ABB RAPID module: Module1.mod

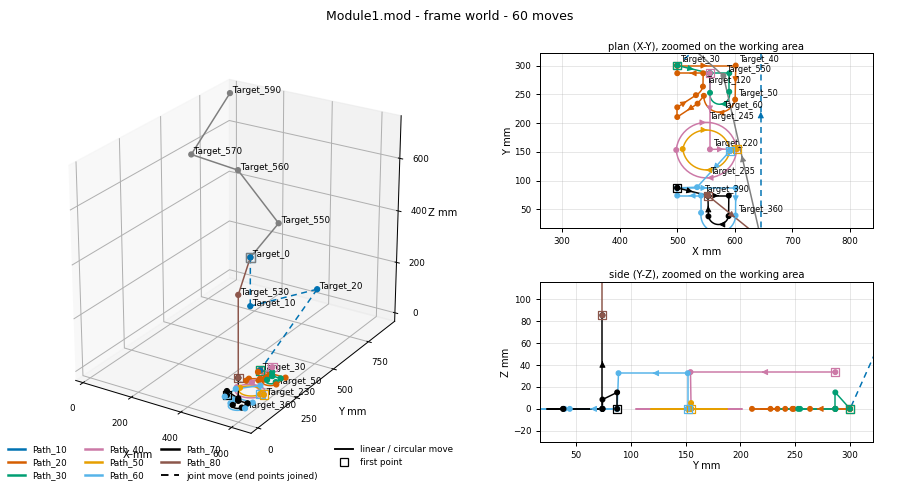
[picture p0: tool path of Module1.mod in frame world, 60 of 60 moves have a stored position in this frame; points joined in program order, loops and branches not executed]
MODULE Module1
    CONST robtarget Target_0:=[[145.114046101,-300,573.947441117],[0.5,0,0.866025404,0],[0,0,0,0],[9E+09,9E+09,9E+09,9E+09,9E+09,9E+09]];
    CONST robtarget Target_10:=[[145.11412777,-300,402.018378698],[0.500000003,0,0.866025402,0],[0,0,0,0],[9E+09,9E+09,9E+09,9E+09,9E+09,9E+09]];
    CONST robtarget Target_20:=[[145.114134181,130.918790149,291.07357],[0.500000009,0.000000018,0.866025398,-0.00000003],[0,-1,1,0],[9E+09,9E+09,9E+09,9E+09,9E+09,9E+09]];
    CONST robtarget Target_30:=[[0,0,0],[0,1,0,0],[0,0,-2,0],[9E+09,9E+09,9E+09,9E+09,9E+09,9E+09]];
    CONST robtarget Target_40:=[[101.558,0,0],[0,1,0,0],[0,0,-2,0],[9E+09,9E+09,9E+09,9E+09,9E+09,9E+09]];
    CONST robtarget Target_50:=[[100.559,-59.146,0],[0,1,0,0],[0,0,-2,0],[9E+09,9E+09,9E+09,9E+09,9E+09,9E+09]];
    CONST robtarget Target_60:=[[73.842,-81.151,0],[0,1,0,0],[0,0,-2,0],[9E+09,9E+09,9E+09,9E+09,9E+09,9E+09]];
    CONST robtarget Target_70:=[[46.206,-52.556,0],[0,1,0,0],[0,0,-2,0],[9E+09,9E+09,9E+09,9E+09,9E+09,9E+09]];
    CONST robtarget Target_80:=[[35.263,-66.215,0],[0,1,0,0],[0,0,-2,0],[9E+09,9E+09,9E+09,9E+09,9E+09,9E+09]];
    CONST robtarget Target_90:=[[-0.001,-89.458,0],[0,1,0,0],[0,0,-2,0],[9E+09,9E+09,9E+09,9E+09,9E+09,9E+09]];
    CONST robtarget Target_100:=[[-0.001,-72.564,0],[0,1,0,0],[0,0,-2,0],[9E+09,9E+09,9E+09,9E+09,9E+09,9E+09]];
    CONST robtarget Target_110:=[[32.467,-51.478,0],[0,1,0,0],[0,0,-2,0],[9E+09,9E+09,9E+09,9E+09,9E+09,9E+09]];
    CONST robtarget Target_115:=[[41.413,-43.371,0],[0,1,0,0],[0,0,-2,0],[9E+09,9E+09,9E+09,9E+09,9E+09,9E+09]];
    CONST robtarget Target_120:=[[44.608,-36.502,0],[0,1,0,0],[0,0,-2,0],[9E+09,9E+09,9E+09,9E+09,9E+09,9E+09]];
    CONST robtarget Target_130:=[[45.087,-13.418,0],[0,1,0,0],[0,0,-2,0],[9E+09,9E+09,9E+09,9E+09,9E+09,9E+09]];
    CONST robtarget Target_140:=[[-0.001,-13.418,0],[0,1,0,0],[0,0,-2,0],[9E+09,9E+09,9E+09,9E+09,9E+09,9E+09]];
    CONST robtarget Target_145:=[[0,0,0],[0,1,0,0],[0,0,-2,0],[9E+09,9E+09,9E+09,9E+09,9E+09,9E+09]];
    CONST robtarget Target_150_IntermedioR:=[[56.636379342,-13.418007291,15.010665058],[-0.000000015,1,0.000000042,0.000000001],[0,0,-2,0],[9E+09,9E+09,9E+09,9E+09,9E+09,9E+09]];
    CONST robtarget Target_150_ZFinal:=[[56.749,-13.418,0],[0,1,0,0],[0,0,-2,0],[9E+09,9E+09,9E+09,9E+09,9E+09,9E+09]];
    CONST robtarget Target_160:=[[90.336,-13.418,0],[0,1,0,0],[0,0,-2,0],[9E+09,9E+09,9E+09,9E+09,9E+09,9E+09]];
    CONST robtarget Target_170:=[[90.336,-45.567,0],[0,1,0,0],[0,0,-2,0],[9E+09,9E+09,9E+09,9E+09,9E+09,9E+09]];
    CONST robtarget Target_180:=[[73.842,-67.293,0],[0,1,0,0],[0,0,-2,0],[9E+09,9E+09,9E+09,9E+09,9E+09,9E+09]];
    CONST robtarget Target_190:=[[56.909,-47.325,0],[0,1,0,0],[0,0,-2,0],[9E+09,9E+09,9E+09,9E+09,9E+09,9E+09]];
    CONST robtarget Target_200:=[[56.749,-13.418,0],[0,1,0,0],[0,0,-2,0],[9E+09,9E+09,9E+09,9E+09,9E+09,9E+09]];
    CONST robtarget Target_210:=[[56.748968334,-13.418012212,33.529365391],[-0.000000004,1,-0.000000052,-0.000000031],[0,0,-2,0],[9E+09,9E+09,9E+09,9E+09,9E+09,9E+09]];
    CONST robtarget Target_220:=[[56.748986906,-145.605410925,33.52934752],[0,1,-0.000000083,-0.000000019],[0,0,-2,0],[9E+09,9E+09,9E+09,9E+09,9E+09,9E+09]];
    CONST robtarget Target_230:=[[103.355,-145.049,0],[0,1,0,0],[0,0,-2,0],[9E+09,9E+09,9E+09,9E+09,9E+09,9E+09]];
    CONST robtarget Target_235:=[[52.116,-195.19,0],[0,1,0,0],[0,0,-2,0],[9E+09,9E+09,9E+09,9E+09,9E+09,9E+09]];
    CONST robtarget Target_240:=[[-1.758,-146.687,0],[0,1,0,0],[0,0,-2,0],[9E+09,9E+09,9E+09,9E+09,9E+09,9E+09]];
    CONST robtarget Target_245:=[[50.261,-98.729,0],[0,1,0,0],[0,0,-2,0],[9E+09,9E+09,9E+09,9E+09,9E+09,9E+09]];
    CONST robtarget Target_250:=[[103.355,-145.049,0],[0,1,0,0],[0,0,-2,0],[9E+09,9E+09,9E+09,9E+09,9E+09,9E+09]];
    CONST robtarget Target_260:=[[97.170116811,-145.0489929,5.322039607],[0.000000004,1,0.000000037,0.000000006],[0,-1,-2,0],[9E+09,9E+09,9E+09,9E+09,9E+09,9E+09]];
    CONST robtarget Target_270:=[[91.773,-147.965,0],[0,1,0,0],[0,0,-2,0],[9E+09,9E+09,9E+09,9E+09,9E+09,9E+09]];
    CONST robtarget Target_280:=[[48.761,-181.312,0],[0,1,0,0],[0,0,-2,0],[9E+09,9E+09,9E+09,9E+09,9E+09,9E+09]];
    CONST robtarget Target_290:=[[9.487,-145.045,0],[0,1,0,0],[0,0,-2,0],[9E+09,9E+09,9E+09,9E+09,9E+09,9E+09]];
    CONST robtarget Target_300:=[[50.519,-112.002,0],[0,1,0,0],[0,0,-2,0],[9E+09,9E+09,9E+09,9E+09,9E+09,9E+09]];
    CONST robtarget Target_310:=[[91.935,-148.087,0],[0,1,0,0],[0,0,-2,0],[9E+09,9E+09,9E+09,9E+09,9E+09,9E+09]];
    CONST robtarget Target_320:=[[91.93496497,-148.087005279,32.547397703],[0.000000003,1,0.000000045,-0.000000008],[0,-1,-2,0],[9E+09,9E+09,9E+09,9E+09,9E+09,9E+09]];
    CONST robtarget Target_330:=[[34.441170169,-211.299624395,32.547366159],[-0.000000002,1,0.000000004,-0.000000023],[0,0,-2,0],[9E+09,9E+09,9E+09,9E+09,9E+09,9E+09]];
    CONST robtarget Target_340:=[[-0.001,-212.542,0],[0,1,0,0],[0,0,-2,0],[9E+09,9E+09,9E+09,9E+09,9E+09,9E+09]];
    CONST robtarget Target_350:=[[101.558,-212.542,0],[0,1,0,0],[0,0,-2,0],[9E+09,9E+09,9E+09,9E+09,9E+09,9E+09]];
    CONST robtarget Target_360:=[[101.278,-260.506,0],[0,1,0,0],[0,0,-2,0],[9E+09,9E+09,9E+09,9E+09,9E+09,9E+09]];
    CONST robtarget Target_370:=[[72.204,-290.019,0],[0,1,0,0],[0,0,-2,0],[9E+09,9E+09,9E+09,9E+09,9E+09,9E+09]];
    CONST robtarget Target_380:=[[41.373,-255.754,0],[0,1,0,0],[0,0,-2,0],[9E+09,9E+09,9E+09,9E+09,9E+09,9E+09]];
    CONST robtarget Target_390:=[[41.293,-225.961,0],[0,1,0,0],[0,0,-2,0],[9E+09,9E+09,9E+09,9E+09,9E+09,9E+09]];
    CONST robtarget Target_400:=[[-0.001,-225.961,0],[0,1,0,0],[0,0,-2,0],[9E+09,9E+09,9E+09,9E+09,9E+09,9E+09]];
    CONST robtarget Target_410:=[[-0.001,-212.542,0],[0,1,0,0],[0,0,-2,0],[9E+09,9E+09,9E+09,9E+09,9E+09,9E+09]];
    CONST robtarget Target_420:=[[-0.00102366,-212.542012413,15.028104182],[-0.000000001,1,-0.000000059,-0.000000007],[0,0,-2,0],[9E+09,9E+09,9E+09,9E+09,9E+09,9E+09]];
    CONST robtarget Target_430:=[[53.40676855,-225.942037535,8.490466142],[-0.000000001,1,-0.000000385,-0.000000007],[0,0,-2,0],[9E+09,9E+09,9E+09,9E+09,9E+09,9E+09]];
    CONST robtarget Target_440:=[[53.274,-225.961,0],[0,1,0,0],[0,0,-2,0],[9E+09,9E+09,9E+09,9E+09,9E+09,9E+09]];
    CONST robtarget Target_450:=[[89.577,-225.961,0],[0,1,0,0],[0,0,-2,0],[9E+09,9E+09,9E+09,9E+09,9E+09,9E+09]];
    CONST robtarget Target_460:=[[89.177,-261.505,0],[0,1,0,0],[0,0,-2,0],[9E+09,9E+09,9E+09,9E+09,9E+09,9E+09]];
    CONST robtarget Target_470:=[[71.765,-276.161,0],[0,1,0,0],[0,0,-2,0],[9E+09,9E+09,9E+09,9E+09,9E+09,9E+09]];
    CONST robtarget Target_480:=[[54.153,-261.984,0],[0,1,0,0],[0,0,-2,0],[9E+09,9E+09,9E+09,9E+09,9E+09,9E+09]];
    CONST robtarget Target_490:=[[53.274,-225.961,0],[0,1,0,0],[0,0,-2,0],[9E+09,9E+09,9E+09,9E+09,9E+09,9E+09]];
    CONST robtarget Target_500:=[[53.273969687,-225.961003513,85.391501657],[-0.000000001,1,0.000000011,-0.000000007],[0,0,-2,0],[9E+09,9E+09,9E+09,9E+09,9E+09,9E+09]];
    CONST robtarget Target_530:=[[53.273975183,-225.961003543,389.504685045],[0.000000001,1,0.000000014,-0.000000011],[0,0,-2,0],[9E+09,9E+09,9E+09,9E+09,9E+09,9E+09]];
    CONST robtarget Target_540:=[[145.114046101,-300,573.947441117],[0.5,0,0.866025404,0],[0,0,0,0],[9E+09,9E+09,9E+09,9E+09,9E+09,9E+09]];
    CONST robtarget Target_550:=[[80.158887002,-17.886905109,573.947441117],[0.487251492,-0.194314053,0.84394434,0.112187271],[0,0,0,0],[9E+09,9E+09,9E+09,9E+09,9E+09,9E+09]];
    CONST robtarget Target_560:=[[-281.152242484,306.8589552,573.947441117],[0.409151388,-0.497780499,0.708670992,0.287393705],[0,-1,-1,0],[9E+09,9E+09,9E+09,9E+09,9E+09,9E+09]];
    CONST robtarget Target_570:=[[-500.572509967,345.113792062,573.947441117],[0.353396474,-0.612644102,0.612100649,0.353710237],[1,-1,0,0],[9E+09,9E+09,9E+09,9E+09,9E+09,9E+09]];
    CONST robtarget Target_590:=[[-500.801741318,603.468233425,725.305628398],[0.499667188,-0.50033274,0.499889039,0.500110787],[1,-1,0,0],[9E+09,9E+09,9E+09,9E+09,9E+09,9E+09]];
    PROC Path_10()
        MoveJ Target_0,v1000,z10,ChuislitoToolTCP\WObj:=TablaPlana;
        MoveJ Target_10,v1000,z10,ChuislitoToolTCP\WObj:=TablaPlana;
        MoveJ Target_20,v1000,z10,ChuislitoToolTCP\WObj:=TablaPlana;
        MoveJ Target_30,v1000,z10,ChuislitoToolTCP\WObj:=TablaPlana;
    ENDPROC
    PROC Path_20()
        MoveL Target_30,v100,z5,ChuislitoToolTCP\WObj:=TablaPlana;
        MoveL Target_40,v100,z5,ChuislitoToolTCP\WObj:=TablaPlana;
        MoveL Target_50,v100,z5,ChuislitoToolTCP\WObj:=TablaPlana;
        MoveC Target_60,Target_70,v100,z5,ChuislitoToolTCP\WObj:=TablaPlana;
        MoveL Target_80,v100,z5,ChuislitoToolTCP\WObj:=TablaPlana;
        MoveL Target_90,v100,z5,ChuislitoToolTCP\WObj:=TablaPlana;
        MoveL Target_100,v100,z5,ChuislitoToolTCP\WObj:=TablaPlana;
        MoveL Target_110,v100,z5,ChuislitoToolTCP\WObj:=TablaPlana;
        MoveC Target_115,Target_120,v100,z5,ChuislitoToolTCP\WObj:=TablaPlana;
        MoveL Target_130,v100,z5,ChuislitoToolTCP\WObj:=TablaPlana;
        MoveL Target_140,v100,z5,ChuislitoToolTCP\WObj:=TablaPlana;
        MoveL Target_145,v100,z5,ChuislitoToolTCP\WObj:=TablaPlana;
    ENDPROC
    PROC Path_30()
        MoveL Target_145,v100,z5,ChuislitoToolTCP\WObj:=TablaPlana;
        MoveL Target_150_IntermedioR,v100,z5,ChuislitoToolTCP\WObj:=TablaPlana;
        MoveL Target_150_ZFinal,v100,z5,ChuislitoToolTCP\WObj:=TablaPlana;
        MoveL Target_160,v100,z5,ChuislitoToolTCP\WObj:=TablaPlana;
        MoveL Target_170,v100,z5,ChuislitoToolTCP\WObj:=TablaPlana;
        MoveC Target_180,Target_190,v100,z5,ChuislitoToolTCP\WObj:=TablaPlana;
        MoveL Target_200,v100,z5,ChuislitoToolTCP\WObj:=TablaPlana;
    ENDPROC
    PROC Path_40()
        MoveL Target_210,v100,z5,ChuislitoToolTCP\WObj:=TablaPlana;
        MoveL Target_220,v100,z5,ChuislitoToolTCP\WObj:=TablaPlana;
        MoveL Target_230,v100,z5,ChuislitoToolTCP\WObj:=TablaPlana;
        MoveC Target_235,Target_240,v100,z5,ChuislitoToolTCP\WObj:=TablaPlana;
        MoveC Target_245,Target_250,v100,z5,ChuislitoToolTCP\WObj:=TablaPlana;
    ENDPROC
    PROC Path_50()
        MoveL Target_250,v100,z5,ChuislitoToolTCP\WObj:=TablaPlana;
        MoveL Target_260,v100,z5,ChuislitoToolTCP\WObj:=TablaPlana;
        MoveL Target_270,v100,z5,ChuislitoToolTCP\WObj:=TablaPlana;
        MoveC Target_280,Target_290,v100,z5,ChuislitoToolTCP\WObj:=TablaPlana;
        MoveC Target_300,Target_310,v100,z5,ChuislitoToolTCP\WObj:=TablaPlana;
    ENDPROC
    PROC Path_60()
        MoveL Target_310,v100,z5,ChuislitoToolTCP\WObj:=TablaPlana;
        MoveL Target_320,v100,z5,ChuislitoToolTCP\WObj:=TablaPlana;
        MoveL Target_330,v100,z5,ChuislitoToolTCP\WObj:=TablaPlana;
        MoveL Target_340,v100,z5,ChuislitoToolTCP\WObj:=TablaPlana;
        MoveL Target_350,v100,z5,ChuislitoToolTCP\WObj:=TablaPlana;
        MoveL Target_360,v100,z5,ChuislitoToolTCP\WObj:=TablaPlana;
        MoveC Target_370,Target_380,v100,z5,ChuislitoToolTCP\WObj:=TablaPlana;
        MoveL Target_390,v100,z5,ChuislitoToolTCP\WObj:=TablaPlana;
        MoveL Target_400,v100,z5,ChuislitoToolTCP\WObj:=TablaPlana;
        MoveL Target_410,v100,z5,ChuislitoToolTCP\WObj:=TablaPlana;
    ENDPROC
    PROC Path_70()
        MoveL Target_410,v100,z5,ChuislitoToolTCP\WObj:=TablaPlana;
        MoveL Target_420,v100,z5,ChuislitoToolTCP\WObj:=TablaPlana;
        MoveL Target_430,v100,z5,ChuislitoToolTCP\WObj:=TablaPlana;
        MoveL Target_440,v100,z5,ChuislitoToolTCP\WObj:=TablaPlana;
        MoveL Target_450,v100,z5,ChuislitoToolTCP\WObj:=TablaPlana;
        MoveL Target_460,v100,z5,ChuislitoToolTCP\WObj:=TablaPlana;
        MoveC Target_470,Target_480,v100,z5,ChuislitoToolTCP\WObj:=TablaPlana;
        MoveL Target_490,v100,z5,ChuislitoToolTCP\WObj:=TablaPlana;
        MoveL Target_500,v100,z5,ChuislitoToolTCP\WObj:=TablaPlana;
    ENDPROC
    PROC Path_80()
        MoveL Target_500,v100,z5,ChuislitoToolTCP\WObj:=TablaPlana;
        MoveL Target_530,v100,z5,ChuislitoToolTCP\WObj:=TablaPlana;
        MoveL Target_540,v100,z5,ChuislitoToolTCP\WObj:=TablaPlana;
    ENDPROC
    PROC mantenimiento()
        MoveL Target_540,v100,z5,ChuislitoToolTCP\WObj:=TablaPlana;
        MoveL Target_550,v100,z5,ChuislitoToolTCP\WObj:=TablaPlana;
        MoveL Target_560,v100,z5,ChuislitoToolTCP\WObj:=TablaPlana;
        MoveL Target_570,v100,z5,ChuislitoToolTCP\WObj:=TablaPlana;
        MoveL Target_590,v100,z5,ChuislitoToolTCP\WObj:=TablaPlana;
    ENDPROC

    PROC main()
        WHILE EntDI_2 = 0 OR EntDI_1= 0 DO
        IF EntDI_2=1 THEN
             SetDO SalDO_1,0;
             mantenimiento;
        ELSEIF EntDI_1=1 THEN
            SetDO SalDO_1,1;
            Path_10;
            Path_20;
            Path_30;
            Path_40;
            Path_50;
            Path_60;
            Path_70;
            Path_80;
        ELSE
            SetDO SalDO_1,0;
        ENDIF
        ENDWHILE
    ENDPROC

ENDMODULE
